// TIA Portal V20 export
DATA_BLOCK "GDB_MCDData"   // DB6
{ S7_Optimized_Access := 'TRUE' }
// stored: MemoryReserve 100
   VAR
      Velocity : Array[1..4] of LReal;   // Kinematic-group view of per-axis velocity (from ScaraArm3D.AxesData.A[i].Velocity). Used by NX MCD via signal adapters.
      Position : Array[1..4] of LReal;   // Kinematic-group view of per-axis position (from ScaraArm3D.AxesData.A[i].Position). Used by NX MCD via signal adapters.
      J1_ActualPosition : LReal;   // Phase C.0 (2026-05-17): direct mirror of J1_SCARA_Arm3D.ActualPosition (TO_Axis attribute). Exists for PLCSIM-Adv API monitoring (TO_Axis tags not exposed via API directly; HMI runtime uses TIA S7 driver which can read them). DIAGNOSTIC MIRROR — HMI continues to bind to J1_SCARA_Arm3D.ActualPosition direct.
      J1_ActualVelocity : LReal;   // Phase C.0 (2026-05-17): direct mirror of J1_SCARA_Arm3D.ActualVelocity. See J1_ActualPosition comment.
      J2_ActualPosition : LReal;   // Phase C.0 (2026-05-17): direct mirror of J2_SCARA_Arm3D.ActualPosition. See J1_ActualPosition comment.
      J2_ActualVelocity : LReal;   // Phase C.0 (2026-05-17): direct mirror of J2_SCARA_Arm3D.ActualVelocity. See J1_ActualPosition comment.
      J3_ActualPosition : LReal;   // Phase C.0 (2026-05-17): direct mirror of J3_SCARA_Arm3D.ActualPosition. See J1_ActualPosition comment.
      J3_ActualVelocity : LReal;   // Phase C.0 (2026-05-17): direct mirror of J3_SCARA_Arm3D.ActualVelocity. See J1_ActualPosition comment.
      J4_ActualPosition : LReal;   // Phase C.0 (2026-05-17): direct mirror of J4_SCARA_Arm3D.ActualPosition. See J1_ActualPosition comment.
      J4_ActualVelocity : LReal;   // Phase C.0 (2026-05-17): direct mirror of J4_SCARA_Arm3D.ActualVelocity. See J1_ActualPosition comment.
   END_VAR
BEGIN
END_DATA_BLOCK
